PROGRAM Axis03_Status
VAR
//System_Bit
	Always_ON	:	BOOL	:=TRUE	;//상시 ON 
	Always_OFF	:	BOOL	:=FALSE	;//상시 OFF
	
//Motor_Command
	Axis03_Status_01: MC_ReadStatus;
	Axis03_Position_Read_01: MC_ReadActualPosition;
	Axis03_Velocity_Read_01: MC_ReadActualVelocity;
	Axis03_Reset_01: MC_Reset;
	Axis03_Stop_01: MC_Stop;
END_VAR

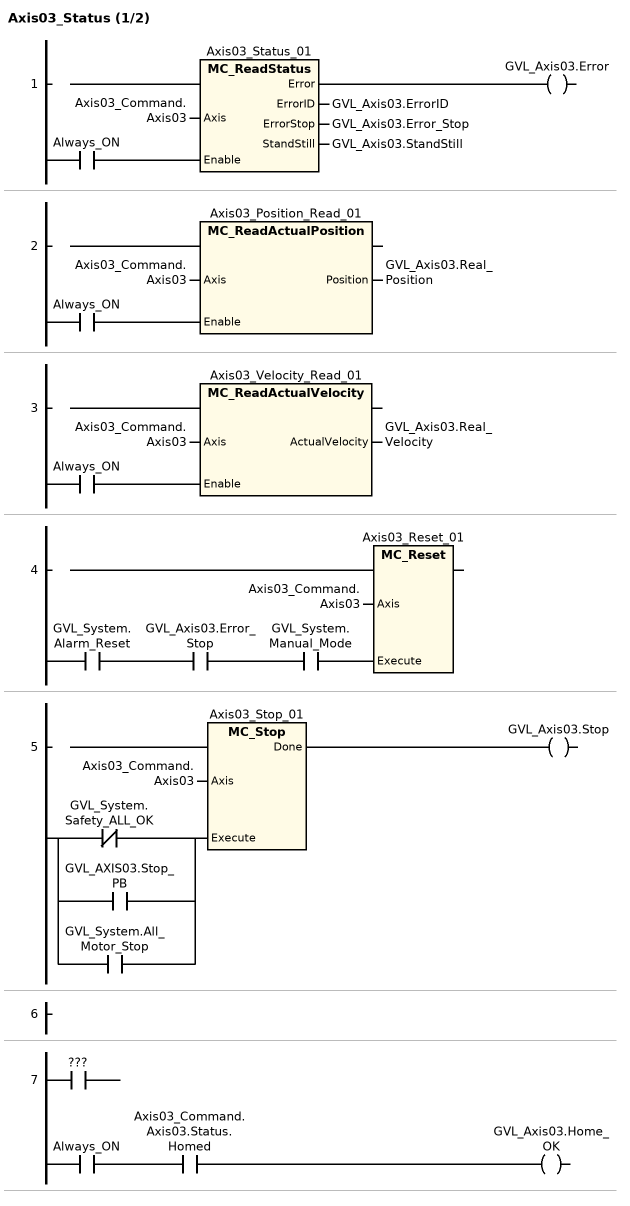
// NETWORK 1
Axis03_Status_01(
    Axis := Axis03_Command.Axis03,
    Enable := Always_ON,
    Error => GVL_Axis03.Error,
    ErrorID => GVL_Axis03.ErrorID,
    ErrorStop => GVL_Axis03.Error_Stop,
    StandStill => GVL_Axis03.StandStill); // MC_ReadStatus

// NETWORK 2
Axis03_Position_Read_01(
    Axis := Axis03_Command.Axis03,
    Enable := Always_ON,
    Position => GVL_Axis03.Real_Position); // MC_ReadActualPosition

// NETWORK 3
Axis03_Velocity_Read_01(
    Axis := Axis03_Command.Axis03,
    Enable := Always_ON,
    ActualVelocity => GVL_Axis03.Real_Velocity); // MC_ReadActualVelocity

// NETWORK 4
Axis03_Reset_01(Axis := Axis03_Command.Axis03, Execute := GVL_System.Alarm_Reset AND GVL_Axis03.Error_Stop AND GVL_System.Manual_Mode); // MC_Reset

// NETWORK 5
Axis03_Stop_01(Axis := Axis03_Command.Axis03, Execute := NOT GVL_System.Safety_ALL_OK OR GVL_AXIS03.Stop_PB OR GVL_System.All_Motor_Stop); // MC_Stop
GVL_Axis03.Stop := Axis03_Stop_01.Done;

// NETWORK 6

// NETWORK 7
GVL_Axis03.Home_OK := Always_ON AND Axis03_Command.Axis03.Status.Homed;

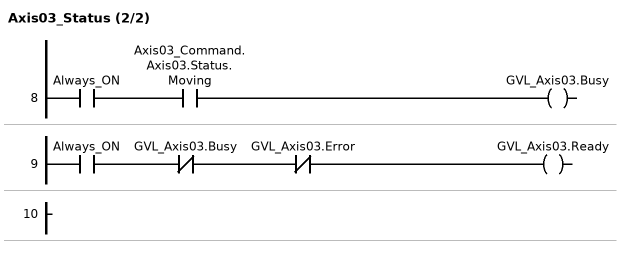
// NETWORK 8
GVL_Axis03.Busy := Always_ON AND Axis03_Command.Axis03.Status.Moving;

// NETWORK 9
GVL_Axis03.Ready := Always_ON AND NOT GVL_Axis03.Busy AND NOT GVL_Axis03.Error;

// NETWORK 10

END_PROGRAM

(* stored: Version 1.1.0.1, ProductVersion 3.1.4024.16
   POU Axis03_Status: Id {6772cf1a-0606-4815-9c2e-28638ae5dcce}, SpecialFunc None *)
